(*			
	RAFALOS
	Rafał Osajda		19.09.2025		TC 4024.66
	
*)
FUNCTION_BLOCK FB_BaseDescriptor IMPLEMENTS ITF_BaseDescriptor
VAR
	stDeskryptor					: ST_Descriptor;
END_VAR

END_FUNCTION_BLOCK

(* stored: Version 1.1.0.1
   POU FB_BaseDescriptor: Id {91493404-5653-0352-2d94-26778011a0ca}, SpecialFunc None *)
